(* IEC 61131-3 sources: stopGate_FuB/Logical/FSM/VT_Infeed/Infeed0, 5 files *)

(* ---- Types.typ ---- *)
TYPE

END_TYPE

(* ---- Cyclic.st ---- *)
PROGRAM _CYCLIC
	//**************************************************************************//
	// VT--> InfeedZone 0 communications****************************************//
	// Sept 6, 2024*************************************************************//
	// Jamie Dukelow, Assurant Inc.*********************************************//
	//**************************************************************************//

	//Handoff between VT and Infeed Zone 0

	bladeStopZone0();
	partPresent := bladeStopZone0.partPresent;
	gateOpen := bladeStopZone0.gateOpen;
	gateClose := bladeStopZone0.gateClose;
	hasOpenSensor := bladeStopZone0.hasOpenSensor;
	downstreamReady := bladeStopZone0.downstreamReady;
	EMGC := bladeStopZone0.EMGC;

END_PROGRAM

(* ---- Exit.st ---- *)
PROGRAM _EXIT
	(* Insert code here *)

END_PROGRAM

(* ---- Init.st ---- *)
PROGRAM _INIT
	(* Insert code here *)

END_PROGRAM

(* ---- Variables.var ---- *)
VAR

END_VAR

VAR CONSTANT

END_VAR
